FUNCTION Convert_BYTE_TO_INT : BOOL
VAR_INPUT
	in : BYTE;
	out : REFERENCE TO INT;
END_VAR
VAR
	converted : INT;
END_VAR

converted := BYTE_TO_INT(in);

IF (INT_TO_BYTE(converted) <> in) THEN
	RETURN;
END_IF

out := converted;
Convert_BYTE_TO_INT := TRUE;

END_FUNCTION

(* stored: Version 1.1.0.1, ProductVersion 3.1.4024.12
   POU Convert_BYTE_TO_INT: Id {9179c7e0-dfdd-4f02-9e37-4e5869fbb927}, SpecialFunc None *)
